(* IEC 61131-3 sources: Industry-PLC-LLM/data/PLCBEAD_repo/PLCBEAD_PLCEmbed-main/PLC-BEAD/Source/GEB/MUX_R4, 1 file *)

(* ---- MUX_R4.ST ---- *)
FUNCTION MUX_R4:REAL

	VAR_INPUT
		IN0 :	REAL;
		IN1 :	REAL;
		IN2 :	REAL;
		IN3 :	REAL;
		A0 :	BOOL;
		A1 :	BOOL;
	END_VAR

	IF A1 THEN
		MUX_R4 := SEL(A0, IN2, IN3);
	ELSE
		MUX_R4 := SEL(A0, IN0, IN1);
	END_IF;

END_FUNCTION

PROGRAM program0
	VAR
		IN0 :	REAL;
		IN1 :	REAL;
		IN2 :	REAL;
		IN3 :	REAL;
		A0 :	BOOL;
		A1 :	BOOL;

		OUT : REAL;
	END_VAR

	OUT := MUX_R4(IN0, IN1, IN2, IN3, A0, A1);

END_PROGRAM
